FUNCTION_BLOCK TransitionController
VAR_INPUT
  done: BOOL;
  error: BOOL;
  error_id: UDINT;
END_VAR
VAR_OUTPUT
  execute_level: BOOL;
  execute_trigger: BOOL;
END_VAR
VAR
  lr_execute: LockingRelay;
  r_execute: R_TRIG;
  _execute: BOOL;
  lr_done: LockingRelay;
  lr_error: LockingRelay;
END_VAR

METHOD fire
VAR_INPUT
  execute: BOOL;
END_VAR
lr_execute.clk := execute;
r_execute(CLK:=execute);
IF r_execute.Q THEN
  _execute := TRUE;
END_IF

execute_trigger := r_execute.q;

execute_level := lr_execute.q;
END_METHOD

PROPERTY transition : BOOL
GET
IF _execute THEN
  lr_done.clk := done;
END_IF
lr_error.clk := (error_id <> 0) OR error;
transition := lr_done.q AND NOT lr_error.q;
IF transition THEN
  lr_done.reset := TRUE;
  lr_error.reset := TRUE;
  _execute := FALSE;
END_IF
END_GET
END_PROPERTY

END_FUNCTION_BLOCK

(* stored: Version 1.1.0.1, ProductVersion 3.1.4022.18
   POU TransitionController: Id {20cd3498-8cad-479f-bb2a-eeea5268535f}, SpecialFunc None
   Method fire: Id {0ee15a7f-e0e2-4170-9e85-128b4e88acf2}
   Property transition: Id {9d02efc4-fa97-4c6a-b58b-9f30072c6301}
   Get Get: Id {23c50a87-ec95-474a-a1b2-d6b30d55b759} *)
